(* IEC 61131-3 sources: AXOpen/src/components.siem.identification/app/src/Documentation, 5 files *)

(* ---- Component_1.st ---- *)
USING AXOpen.Core;
USING AXOpen.Components.Siem.Identification;
USING System.Strings;

NAMESPACE AXOpen.Components.Siem.Identification
    {S7.extern=ReadWrite}
    CLASS Component_1 EXTENDS AXOpen.Core.AxoObject
        //<ComponentDeclaration>
        VAR PUBLIC
            IdentProfileReader : AXOpen.Components.Siem.Identification.Axo_IdentDevice;
        END_VAR
        //</ComponentDeclaration>

        //<InitializationArgumentsDeclaration>
        VAR PUBLIC
            {#ix-set:AttributeName = "<#Activate manual control#>"}
            ActivateManualControl : BOOL;
            //Data used for reset sequence
            //The reader must be reseted after each PLC startup
            //For different reader type/family change the reset data according to manual
            //Manual Entry ID: 109793329, Entry date: 02/18/2021
            //Document ID number:	C79000-G8976-C387-06
            //Link: https://cache.industry.siemens.com/dl/files/329/109793329/att_1054102/v1/FH_Ident-Profil_76_en-US.pdf
            //Chapter: 3.5 Programming the Ident profile
            //Page: 80+
            {#ix-attr:[CompilerOmits()]}
            ExampleReader_hardwareConfig: ARRAY[0..15] OF BYTE := [BYTE#16#04,BYTE#16#00,BYTE#16#00,BYTE#16#00,BYTE#16#00,BYTE#16#0A,BYTE#16#00,BYTE#16#00,BYTE#16#00,BYTE#16#25,BYTE#16#00,BYTE#16#00,BYTE#16#00,BYTE#16#01,BYTE#16#00,BYTE#16#01]; //default data for RF260R
            DoNotRun    :   BOOL    :=  FALSE;
        END_VAR
        //</InitializationArgumentsDeclaration>

        METHOD PUBLIC Run
            VAR_INPUT
                parent : IAxoContext;
            END_VAR

            IF DoNotRun THEN
                RETURN;
            END_IF;

            THIS.InitializeWithContext(parent);

            IF ActivateManualControl THEN
                IdentProfileReader.ActivateManualControl();
            END_IF;

            //<Initialization>
            IdentProfileReader.Config.HardwareConfig.Data := ExampleReader_hardwareConfig;

            //For different reader type/family change the CM_CHANNEL, API, SLOT, SUB_SLOT according to application example
            //Application example Entry ID: 109807653, Entry date: 04/21/2022
            //Link: https://cache.industry.siemens.com/dl/files/653/109807653/att_1101693/v2/109807653_Simatic_Ident_Profinet_Beckhoff_DOC_V10_en.pdf
            //Chapter: 2.3.6.2 CM_CHANNEL, API, SLOT, SUB_SLOT
            //Page: 18
            IdentProfileReader.Run(parent      :=  THIS,
                        HW_ID       :=  HwIdentifiers#rf186c_Reader_1__Reader__HwID,
                        API         :=  DWORD#16#5B00,
                        SLOT 		:=  WORD#2,
                        SUB_SLOT 	:=  WORD#1,
                        CM_CHANNEL  :=  UINT#1);

            //</Initialization>

            THIS.UseInSequencer();

        END_METHOD

        //<Usage>
        VAR PUBLIC
            Sequencer   :   AxoSequencer;
            Steps       :   ARRAY[0..9] OF AXOpen.Core.AxoStep;
            WriteData   :   STRING  :=  'Abcdefgh65421';
            ReadData    :   STRING;
        END_VAR

        METHOD PRIVATE UseInSequencer

            Sequencer.Initialize(THIS);
            Sequencer.Open();
            Sequencer.SequenceMode := eAxoSequenceMode#RunOnce;

            IF(Steps[0].Execute(Sequencer, 'Restore')) THEN
                ActivateManualControl := FALSE;
                IdentProfileReader.Restore();
                Sequencer.MoveNext();
            END_IF;

            IF(Steps[1].Execute(Sequencer, 'Reset reader')) THEN
                IF(IdentProfileReader.ResetReader().IsDone()) THEN
                    Sequencer.MoveNext();
                END_IF;
            END_IF;

            IF(Steps[2].Execute(Sequencer, 'Write')) THEN
                IF(IdentProfileReader.Write(WriteData,DWORD#0,UINT#0).IsDone()) THEN
                    Sequencer.MoveNext();
                END_IF;
            END_IF;

            IF(Steps[3].Execute(Sequencer, 'Read')) THEN
                IF(IdentProfileReader.Read(DWORD#0,TO_UINT(LengthOf(WriteData)),UINT#0,ReadData).IsDone()) THEN
                    Sequencer.MoveNext();
                END_IF;
            END_IF;

            IF(Steps[4].Execute(Sequencer, 'Compare')) THEN
                IF(ReadData=WriteData) THEN
                    Sequencer.MoveNext();
                END_IF;
            END_IF;

            IF(Steps[5].Execute(Sequencer, 'SoftReset')) THEN
                IF(IdentProfileReader.SoftReset().IsDone()) THEN
                    Sequencer.MoveNext();
                END_IF;
            END_IF;

            IF(Steps[6].Execute(Sequencer, 'Reset reader')) THEN
                IF(IdentProfileReader.ResetReader().IsDone()) THEN
                    Sequencer.MoveNext();
                END_IF;
            END_IF;

            IF(Steps[7].Execute(Sequencer, 'Restore')) THEN
                ActivateManualControl := FALSE;
                IdentProfileReader.Restore();
                Sequencer.MoveNext();
            END_IF;

            IF(Steps[8].Execute(Sequencer, 'SEQUENCE DONE')) THEN
                Sequencer.CompleteSequence();
            END_IF;

        END_METHOD

        //</Usage>
    END_CLASS
END_NAMESPACE

(* ---- Component_2.st ---- *)
USING AXOpen.Core;
USING AXOpen.Components.Siem.Identification;
USING System.Strings;

NAMESPACE AXOpen.Components.Siem.Identification
    {S7.extern=ReadWrite}
    CLASS Component_2 EXTENDS AXOpen.Core.AxoObject
        //<ComponentDeclaration>
        VAR PUBLIC
            IOlinkReader : AXOpen.Components.Siem.Identification.AxoIOLink_RF200Device;
        END_VAR
        //</ComponentDeclaration>

        //<InitializationArgumentsDeclaration>
        VAR PUBLIC
            {#ix-set:AttributeName = "<#Activate manual control#>"}
            ActivateManualControl : BOOL;
        END_VAR
        //</InitializationArgumentsDeclaration>

        METHOD PUBLIC OVERRIDE Run
            VAR_INPUT
                inParent : IAxoObject;
            END_VAR

            SUPER.Run(inParent);

            IF ActivateManualControl THEN
                IOlinkReader.ActivateManualControl();
            END_IF;

            //<Initialization>

            IOlinkReader.Run(   inParent    :=  THIS,
                                HW_ID       :=  HwIdentifiers#et200sp_CM_4xIO_Link_RF200_CM_4xIO_Link_V2_2_144I_128O_1_CM_4xIO_Link_V2_2_144I_128O_HwID,
                                portAddr    :=  INT#0,
                                version     :=  USINT#11);

            //</Initialization>

        THIS.UseInSequencer();
        END_METHOD

        //<Usage>
        VAR PUBLIC
            Sequencer   :   AxoSequencer;
            Steps       :   ARRAY[0..10] OF AXOpen.Core.AxoStep;
            WriteData   :   STRING  :=  'My_very_first_attempt_to_use_RF2xx_via_IO-Link_interface';
            ReadData    :   STRING;
        END_VAR

        METHOD PRIVATE UseInSequencer

            Sequencer.Run(THIS);
            Sequencer.Open();
            Sequencer.SequenceMode := eAxoSequenceMode#RunOnce;

            IF(Steps[0].Execute(Sequencer, 'Restore')) THEN
                ActivateManualControl := FALSE;
                IOlinkReader.Restore();
                Sequencer.MoveNext();
            END_IF;

            IF(Steps[1].Execute(Sequencer, 'Write Tag')) THEN
                IF(IOlinkReader.WriteTag(WriteData,WORD#0).IsDone()) THEN
                    Sequencer.MoveNext();
                END_IF;
            END_IF;

            IF(Steps[2].Execute(Sequencer, 'Read Tag')) THEN
                IF(IOlinkReader.ReadTag(WORD#0,TO_WORD(LengthOf(WriteData)),ReadData).IsDone()) THEN
                    Sequencer.MoveNext();
                END_IF;
            END_IF;

            IF(Steps[3].Execute(Sequencer, 'Compare')) THEN
                IF(ReadData=WriteData) THEN
                    Sequencer.MoveNext();
                END_IF;
            END_IF;

            IF(Steps[4].Execute(Sequencer, 'Restore')) THEN
                ActivateManualControl := FALSE;
                IOlinkReader.Restore();
                Sequencer.MoveNext();
            END_IF;

            IF(Steps[5].Execute(Sequencer, 'SEQUENCE DONE')) THEN
                Sequencer.CompleteSequence();
            END_IF;

        END_METHOD

        //</Usage>
    END_CLASS
END_NAMESPACE

(* ---- Component_3.st ---- *)
USING AXOpen.Core;
USING AXOpen.Components.Siem.Identification;
USING System.Strings;

NAMESPACE AXOpen.Components.Siem.Identification
    {S7.extern=ReadWrite}
    CLASS Component_3 EXTENDS AXOpen.Core.AxoObject
        //<ComponentDeclaration>
        VAR PUBLIC
            RF260R : AXOpen.Components.Siem.Identification.AxoSimaticIdentCyclic;
        END_VAR
        //</ComponentDeclaration>

        //<InitializationArgumentsDeclaration>
        VAR PUBLIC
            {#ix-set:AttributeName = "<#Activate manual control#>"}
            ActivateManualControl : BOOL;
            DataBuffer : ARRAY[0..127] OF BYTE;
        END_VAR
        //</InitializationArgumentsDeclaration>

        METHOD PUBLIC OVERRIDE Run
            VAR_INPUT
                parent : IAxoObject;
            END_VAR

            SUPER.Run(parent);

            IF ActivateManualControl THEN
                RF260R.ActivateManualControl();
            END_IF;

            //<Initialization>

            RF260R.Run( parent      :=  THIS,
                        hwID        :=  HwIdentifiers#rf186c_cyc_HwID,
                        Port        :=  eAxoSimaticIdentCyclic_Port#X21,
                        DataBuffer  :=  DataBuffer);

            //</Initialization>

        // THIS.UseInSequencer();
        END_METHOD

        //<Usage>
        VAR PUBLIC
            Sequencer   :   AxoSequencer;
            Steps       :   ARRAY[0..10] OF AXOpen.Core.AxoStep;
            WriteData   :   STRING  :=  'My_very_first_attempt_to_use_RF2xx_via_IO-Link_interface';
            ReadData    :   STRING;
        END_VAR

        METHOD PRIVATE UseInSequencer

            Sequencer.Run(THIS);
            Sequencer.Open();
            Sequencer.SequenceMode := eAxoSequenceMode#RunOnce;

            IF(Steps[0].Execute(Sequencer, 'Restore')) THEN
                ActivateManualControl := FALSE;
                RF260R.Restore();
                Sequencer.MoveNext();
            END_IF;

            IF(Steps[1].Execute(Sequencer, 'Write Tag')) THEN
                IF(RF260R.WriteTagField((*WriteData,WORD#0*)).IsDone()) THEN
                    Sequencer.MoveNext();
                END_IF;
            END_IF;

            IF(Steps[2].Execute(Sequencer, 'Read Tag')) THEN
                IF(RF260R.ReadTagField((*WORD#0,TO_WORD(LengthOf(WriteData)),ReadData*)).IsDone()) THEN
                    Sequencer.MoveNext();
                END_IF;
            END_IF;

            IF(Steps[3].Execute(Sequencer, 'Compare')) THEN
                IF(ReadData=WriteData) THEN
                    Sequencer.MoveNext();
                END_IF;
            END_IF;

            IF(Steps[4].Execute(Sequencer, 'Restore')) THEN
                ActivateManualControl := FALSE;
                RF260R.Restore();
                Sequencer.MoveNext();
            END_IF;

            IF(Steps[5].Execute(Sequencer, 'SEQUENCE DONE')) THEN
                Sequencer.CompleteSequence();
            END_IF;

        END_METHOD

        //</Usage>
    END_CLASS
END_NAMESPACE

(* ---- Component_4.st ---- *)
USING AXOpen.Core;
USING AXOpen.Components.Siem.Identification;
USING System.Strings;
USING System.Serialization;

NAMESPACE AXOpen.Components.Siem.Identification
    {S7.extern=ReadWrite}
    CLASS Component_4 EXTENDS AXOpen.Core.AxoObject
        //<ComponentDeclaration>
        VAR PUBLIC
            RF340R : AXOpen.Components.Siem.Identification.AxoSimaticIdentCyclic;
        END_VAR
        //</ComponentDeclaration>

        //<InitializationArgumentsDeclaration>
        VAR PUBLIC
            {#ix-set:AttributeName = "<#Activate manual control#>"}
            ActivateManualControl : BOOL;
            DataBuffer : ARRAY[0..127] OF BYTE;
            TestTagUID : ARRAY[0..7] OF BYTE := [BYTE#224,BYTE#8,BYTE#1,BYTE#215,BYTE#229,BYTE#70,BYTE#94,BYTE#82];
        END_VAR
        //</InitializationArgumentsDeclaration>

        METHOD PUBLIC OVERRIDE Run
            VAR_INPUT
                parent : IAxoObject;
            END_VAR

            SUPER.Run(parent);

            IF ActivateManualControl THEN
                RF340R.ActivateManualControl();
            END_IF;

            //<Initialization>

            RF340R.Run( parent      :=  THIS,
                        hwID        :=  HwIdentifiers#rf186c_cyc_HwID,
                        Port        :=  eAxoSimaticIdentCyclic_Port#X22,
                        DataBuffer  :=  DataBuffer);

            //</Initialization>

        THIS.UseInSequencer();
        END_METHOD

        //<Usage>
        VAR PUBLIC
            Sequencer   :   AxoSequencer;
            Steps       :   ARRAY[0..11] OF AXOpen.Core.AxoStep;
            WriteData   :   STRING  :=  'My_very_first_attempt_to_use_RF340Rwith_RF186C_using_cyclic_communication_tag_field_10lenght100bytes';
            ReadData    :   STRING;
        END_VAR

        METHOD PRIVATE UseInSequencer
            VAR
                _index      :   UINT;
                _is_equal   :   BOOL;
                _data       :   ARRAY[0..128] OF BYTE;
                _offset     :   UDINT;
            END_VAR

            Sequencer.Run(THIS);
            Sequencer.Open();
            Sequencer.SequenceMode := eAxoSequenceMode#RunOnce;

            IF(Steps[0].Execute(Sequencer, 'Restore')) THEN
                ActivateManualControl := FALSE;
                RF340R.Restore();
                Sequencer.MoveNext();
            END_IF;

            IF(Steps[1].Execute(Sequencer, 'Reset')) THEN
                IF(RF340R.Reset().IsDone()) THEN
                    Sequencer.MoveNext();
                END_IF;
            END_IF;

            IF(Steps[2].Execute(Sequencer, 'ReadUID')) THEN
                IF(RF340R.ReadUID().IsDone()) THEN
                    Sequencer.MoveNext();
                END_IF;
            END_IF;

            IF(Steps[3].Execute(Sequencer, 'Compare UID')) THEN
                _is_equal := TRUE;
                FOR _index := UINT#0 TO UINT#7 BY UINT#1 DO
                    IF DataBuffer[_index] <> TestTagUID[_index] THEN
                        _is_equal := FALSE;
                    END_IF;
                END_FOR;
                IF(_is_equal) THEN
                    Sequencer.MoveNext();
                END_IF;
            END_IF;

            //  Tag with ID 10 and length 100 has to be already defined using WBM
            IF(Steps[4].Execute(Sequencer, 'WriteTagField: 10, length 100')) THEN
                //*******************************************************************************************//
                // Serialization of the string to the array of bytes to get out its length at the _data[0]
                    _offset := Serialize(UDINT#0, WriteData, _data);
                    FOR _index := UINT#0 TO TO_UINT(_offset) - UINT#1 BY UINT#1 DO
                        DataBuffer[_index] := _data[_index + UINT#1];
                    END_FOR;
                //*******************************************************************************************//
                IF(RF340R.WriteTagField(TagField := UINT#10, TagFieldLength := UINT#100).IsDone()) THEN
                    Sequencer.MoveNext();
                END_IF;
            END_IF;

            //  Tag with ID 10 and length 100 has to be already defined using WBM
            IF(Steps[5].Execute(Sequencer, 'ReadTagField: 10')) THEN
                IF(RF340R.ReadTagField(TagField := UINT#10).IsDone()) THEN
                    Sequencer.MoveNext();
                END_IF;
            END_IF;

            IF(Steps[6].Execute(Sequencer, 'Compare TagField')) THEN
                //*******************************************************************************************//
                // Deserialization of the string from the array of bytes to get its length at the _data[0]
                _data[0] := BYTE#100;
                FOR _index := UINT#0 TO TO_UINT(_offset) - UINT#1 BY UINT#1 DO
                    _data[_index + UINT#1] := DataBuffer[_index];
                END_FOR;

                _offset := Deserialize(UDINT#0,_data, ReadData );
                //*******************************************************************************************//
                IF(ReadData = WriteData) THEN
                    Sequencer.MoveNext();
                END_IF;
            END_IF;

            IF(Steps[7].Execute(Sequencer, 'Write: address: 10, length 8')) THEN
                DataBuffer[0] := BYTE#10;
                DataBuffer[1] := BYTE#20;
                DataBuffer[2] := BYTE#30;
                DataBuffer[3] := BYTE#40;
                DataBuffer[4] := BYTE#50;
                DataBuffer[5] := BYTE#60;
                DataBuffer[6] := BYTE#70;
                DataBuffer[7] := BYTE#80;
                IF(RF340R.Write(Address := UDINT#10, Length := UINT#8).IsDone()) THEN
                    DataBuffer[0] := BYTE#0;
                    DataBuffer[1] := BYTE#0;
                    DataBuffer[2] := BYTE#0;
                    DataBuffer[3] := BYTE#0;
                    DataBuffer[4] := BYTE#0;
                    DataBuffer[5] := BYTE#0;
                    DataBuffer[6] := BYTE#0;
                    DataBuffer[7] := BYTE#0;
                    Sequencer.MoveNext();
                END_IF;
            END_IF;

            IF(Steps[8].Execute(Sequencer, 'Read: address: 10, length 8')) THEN
                IF(RF340R.Read(Address := UDINT#10, Length := UINT#8).IsDone()) THEN
                    Sequencer.MoveNext();
                END_IF;
            END_IF;

            IF(Steps[9].Execute(Sequencer, 'Compare')) THEN
                _is_equal :=    DataBuffer[0] = BYTE#10 AND
                                DataBuffer[1] = BYTE#20 AND
                                DataBuffer[2] = BYTE#30 AND
                                DataBuffer[3] = BYTE#40 AND
                                DataBuffer[4] = BYTE#50 AND
                                DataBuffer[5] = BYTE#60 AND
                                DataBuffer[6] = BYTE#70 AND
                                DataBuffer[7] = BYTE#80;
                IF _is_equal THEN
                    Sequencer.MoveNext();
                END_IF;
            END_IF;

            IF(Steps[10].Execute(Sequencer, 'Restore')) THEN
                ActivateManualControl := FALSE;
                RF340R.Restore();
                Sequencer.MoveNext();
            END_IF;

            IF(Steps[11].Execute(Sequencer, 'SEQUENCE DONE')) THEN
                Sequencer.CompleteSequence();
            END_IF;
        END_METHOD

        //</Usage>
    END_CLASS
END_NAMESPACE

(* ---- DocumentationContext.st ---- *)
NAMESPACE AXOpen.Components.Siem.Identification

    {S7.extern=ReadWrite}
    CLASS DocumentationContext EXTENDS AXOpen.Core.AxoContext
        VAR PUBLIC
            _rootObject     :   AxoObject;
            componentOne    :   Component_1;
            componentTwo    :   Component_2;
            componentThree  :   Component_3;
            componentFour   :   Component_4;
        END_VAR

        METHOD PROTECTED OVERRIDE Main
            THIS.InitializeRootObject(_rootObject);
            componentOne.Run(_rootObject);
            componentTwo.Run(_rootObject);
            componentThree.Run(_rootObject);
            componentFour.Run(_rootObject);
        END_METHOD
    END_CLASS
END_NAMESPACE
